FUNCTION_BLOCK Object IMPLEMENTS I_Object
VAR
	_Name : T_MaxString;
END_VAR

//FB_Init is always available implicitly and it is used primarily for initialization.
//The return value is not evaluated. For a specific influence, you can also declare the
//methods explicitly and provide additional code there with the standard initialization
//code. You can evaluate the return value.
METHOD FB_Init: BOOL
VAR_INPUT
    bInitRetains: BOOL; // TRUE: the retain variables are initialized (reset warm / reset cold)
    bInCopyCode: BOOL;  // TRUE: the instance will be copied to the copy code afterward (online change)  
	Name : T_MaxString; 
END_VAR
_Name := Name;
END_METHOD

PROPERTY Name : T_MaxString
GET
END_GET
END_PROPERTY

METHOD RegisterWithParent
VAR_INPUT
	Parent	: I_HostObjects;
END_VAR
END_METHOD

END_FUNCTION_BLOCK

(* stored: Version 1.1.0.1
   POU Object: Id {3eef5c14-dd0e-4f43-be11-a2e50aecaa97}, SpecialFunc None
   Method FB_Init: Id {0aadef3a-e355-48c1-a003-fae3f4f24a87}
   Property Name: Id {dbd74e7a-7a0a-4226-bf67-82c248c72d59}
   Get Get: Id {31e44081-b98e-4ec8-bc6c-b288dc6ac869}
   Method RegisterWithParent: Id {2bc4b5ec-e7e6-4315-a2f9-26505d5239bf} *)
